//{attribute 'qualified_only'}
{attribute 'strict'}
TYPE E_StateDevice :
(
	eOn      := 0,
	eOff     := 1,
	eForward := 2,
	eReverse := 3,
	eReset   := 4,
	eFault   := 5,
	eAuto    := 6
);
END_TYPE

(* stored: Version 1.1.0.1, ProductVersion 3.1.4024.12
   EnumerationTextList E_StateDevice: Id {36aaf867-59fd-43c0-8f9e-3c95455ffa1d} *)
